FUNCTION_BLOCK FB_TCPModbusRequest
VAR_INPUT
	b_Enable: BOOL;
	str_IPAdress: STRING(15);
	
		
END_VAR
VAR_OUTPUT
	lreal_RealPower_kW:LREAL;
	lreal_Voltage_L1L2_V: LREAL;
	lreal_Voltage_L2L3_V: LREAL;
	lreal_Voltage_L3L1_V: LREAL;
	lreal_Voltage_L1_V: LREAL;
	lreal_Voltage_L2_V: LREAL;
	lreal_Voltage_L3_V: LREAL;
	lreal_Current_L1_A: LREAL;
	lreal_Current_L2_A: LREAL;
	lreal_Current_L3_A: LREAL;
	lreal_PeakPowerDay_kW: LREAL;
	lreal_Power2_kW: LREAL;
	lreal_ReactivePower_kVAr: LREAL;
	lreal_PowerFactor: LREAL;
	lreal_Frequency_Hz: LREAL;
	lreal_Efficiency: LREAL;
	lreal_InternalTemperature_C: LREAL;
	lreal_IsolationResistance_MOhm: LREAL;
	b_MeterOnline: BOOL;
	lreal_GridVoltage_L1L2_V: LREAL;
	lreal_GridVoltage_L2L3_V: LREAL;
	lreal_GridVoltage_L3L1_V: LREAL;
	lreal_GridVoltage_L1_V: LREAL;
	lreal_GridVoltage_L2_V: LREAL;
	lreal_GridVoltage_L3_V: LREAL;
	lreal_GridCurrent_L1_A: LREAL;
	lreal_GridCurrent_L2_A: LREAL;
	lreal_GridCurrent_L3_A: LREAL;
	lreal_GridPower_kW: LREAL;
	lreal_GridReactivePower_kVAr: LREAL;
	lreal_GridPowerFactor: LREAL;
	lreal_GridFrequency_Hz: LREAL;
	lreal_GridEnergyDelivered_kWh: LREAL;
	lreal_GridEnergySupllied_kWh: LREAL;
	
END_VAR
VAR
	i_State:INT;
	FB_SocketConnect : FB_SocketConnect;
	hSocket : T_HSOCKET;
	FB_SocketSend : FB_SocketSend;
	FB_SocketReceive : FB_SocketReceive;
	byteSendString : ARRAY[1..12] OF BYTE;
	byteSendString_2 : ARRAY[1..12] OF BYTE;
	FB_CloseSockets: FB_SocketCloseAll;
	
	ton_TimeOut: Ton;
	ton_WaitforReconnect: Ton;
	ton_ConnectionEstablised: Ton;
	time_ReconnectTime:TIME:=T#30M;
	b_configured: BOOL;
	byteReceiveString : ARRAY[1..200] OF BYTE;
	FB_BYTE_TO_WORD_1 : FB_CV_BYTE_TO_WORD;
	FB_BYTE_TO_WORD_2 : FB_CV_BYTE_TO_WORD;
	FB_BYTE_TO_WORD_Test1 : FB_CV_BYTE_TO_WORD;
	FB_BYTE_TO_WORD_Test2 : FB_CV_BYTE_TO_WORD;
	FB_WORD_TO_INT : FB_CV_WORD_TO_INT;
	ton_WaitforNetxtRequest: Ton;
	ton_Wait: Ton;
	int_SuccessCounter: INT;
	int_ReconnectCounter: INT;
	int_ErrorCount: INT;
	fbConvertWordToDword		: FB_CV_WORD_TO_DWORD;			//Convert Word to Dword
	fbConvertWordToDint			:	FB_CV_WORD_TO_DINT;
	fb_ConvertBytesToLreal		:fb_Convert4BytesToLreal;
	word1: WORD;
	x: INT;
END_VAR





IF NOT b_Enable THEN			// go to state 0 if not enabled
	i_State := 0;
END_IF


CASE i_State OF
	0:	// wait for enable state
		IF b_Enable THEN
			i_State := 1;
		END_IF
		FB_SocketConnect.bExecute := FALSE;
		FB_SocketSend.bExecute := FALSE;
		FB_SocketSend.bExecute := FALSE;
		ton_TimeOut.IN :=FALSE;	
		ton_ConnectionEstablised.IN := FALSE;
	

	1: // check if configured
		IF b_configured = FALSE THEN
			// request FC3, Register 32064, 25 Words 
			byteSendString[1] := 0;
			byteSendString[2] := 1;
			byteSendString[3] := 0;
			byteSendString[4] := 0;
			byteSendString[5] := 0;
			byteSendString[6] := 6;
			byteSendString[7] := 1;
			byteSendString[8] := 3;
			byteSendString[9] := 125;
			byteSendString[10] := 64;
			byteSendString[11] := 0;
			byteSendString[12] := 25;

			// request FC3, Register 37100 16#90EC, 25 Words 
			byteSendString_2[1] := 0;
			byteSendString_2[2] := 1;
			byteSendString_2[3] := 0;
			byteSendString_2[4] := 0;
			byteSendString_2[5] := 0;
			byteSendString_2[6] := 6;
			byteSendString_2[7] := 1;
			byteSendString_2[8] := 3;
			byteSendString_2[9] := 16#90;
			byteSendString_2[10] := 16#EC;
			byteSendString_2[11] := 0;
			byteSendString_2[12] := 38;
		
			b_configured := TRUE;
		END_IF
		i_State := i_State+1;
		
	2: // open socket
		FB_SocketConnect.bExecute := TRUE;
		ton_TimeOut.IN :=TRUE;
		i_State := i_State+1;
		
	3: // wait for connection established	
		IF NOT FB_SocketConnect.bBusy AND NOT FB_SocketConnect.bError THEN
			ton_TimeOut.IN :=FALSE;
			ton_ConnectionEstablised.IN := TRUE;
			i_State := i_State+1;
		ELSIF FB_SocketConnect.bError OR ton_TimeOut.Q THEN
			ton_TimeOut.IN :=FALSE;
			i_State := 100;
		END_IF
	
	4: //connection established, request data
		ton_Wait.IN := TRUE;
		FB_SocketSend.pSrc:= ADR( byteSendString ); 
			IF ton_Wait.Q THEN
			FB_SocketSend.bExecute := TRUE;
			ton_TimeOut.IN :=TRUE;
			ton_Wait.IN := FALSE;
			i_State := i_State+1;
		END_IF
	
	5: // wait for request sent
		IF NOT FB_SocketSend.bBusy AND NOT FB_SocketSend.bError THEN
			ton_TimeOut.IN :=FALSE;
			FB_SocketSend.bExecute := FALSE;
			i_State := i_State+1;  
		ELSIF FB_SocketSend.bError OR ton_TimeOut.Q THEN
			FB_SocketSend.bExecute := FALSE;
			ton_TimeOut.IN :=FALSE;
			i_State := 100;
		END_IF
		
	6: // wait for data
		ton_Wait.IN := TRUE;
		IF ton_Wait.Q THEN
			FB_SocketReceive.bExecute := TRUE;
			ton_Wait.IN := FALSE;
			i_State := i_State+1; 
		END_IF		 
	
	7:	
		ton_Wait.IN := TRUE;
		IF ton_Wait.Q THEN
			ton_TimeOut.IN :=TRUE;
			i_State := i_State+1; 
		END_IF	
	
	8: // convert received data
		IF NOT FB_SocketReceive.bBusy AND NOT FB_SocketReceive.bError THEN
			int_SuccessCounter := int_SuccessCounter+1;
			ton_TimeOut.IN :=FALSE;
			FB_SocketReceive.bExecute := FALSE;
	
			FB_BYTE_TO_WORD_1(byInputValue_1 := byteReceiveString[14],byInputValue_2 := byteReceiveString[15], Ebyteorderforconvert := Ebyteorder.EBIGENDIAN, woutputvalue => );
			lreal_Voltage_L1L2_V := WORD_TO_LREAL(FB_BYTE_TO_WORD_1.woutputvalue)/10;
			FB_BYTE_TO_WORD_1(byInputValue_1 := byteReceiveString[16],byInputValue_2 := byteReceiveString[17], Ebyteorderforconvert := Ebyteorder.EBIGENDIAN, woutputvalue => );
			lreal_Voltage_L2L3_V := WORD_TO_LREAL(FB_BYTE_TO_WORD_1.woutputvalue)/10;
			FB_BYTE_TO_WORD_1(byInputValue_1 := byteReceiveString[18],byInputValue_2 := byteReceiveString[19], Ebyteorderforconvert := Ebyteorder.EBIGENDIAN, woutputvalue => );
			lreal_Voltage_L3L1_V := WORD_TO_LREAL(FB_BYTE_TO_WORD_1.woutputvalue)/10;
			FB_BYTE_TO_WORD_1(byInputValue_1 := byteReceiveString[20],byInputValue_2 := byteReceiveString[21], Ebyteorderforconvert := Ebyteorder.EBIGENDIAN, woutputvalue => );
			lreal_Voltage_L1_V := WORD_TO_LREAL(FB_BYTE_TO_WORD_1.woutputvalue)/10;
			FB_BYTE_TO_WORD_1(byInputValue_1 := byteReceiveString[22],byInputValue_2 := byteReceiveString[23], Ebyteorderforconvert := Ebyteorder.EBIGENDIAN, woutputvalue => );
			lreal_Voltage_L2_V := WORD_TO_LREAL(FB_BYTE_TO_WORD_1.woutputvalue)/10;
			FB_BYTE_TO_WORD_1(byInputValue_1 := byteReceiveString[24],byInputValue_2 := byteReceiveString[25], Ebyteorderforconvert := Ebyteorder.EBIGENDIAN, woutputvalue => );
			lreal_Voltage_L3_V := WORD_TO_LREAL(FB_BYTE_TO_WORD_1.woutputvalue)/10;


			fb_ConvertBytesToLreal(	by_InputValue_1:= byteReceiveString[10], 
									by_InputValue_2:= byteReceiveString[11], 
									by_InputValue_3:= byteReceiveString[12], 
									by_InputValue_4:= byteReceiveString[13], 
									int_Divider:= 1000, 
									lreal_Output=> lreal_RealPower_kW);

			fb_ConvertBytesToLreal(	by_InputValue_1:= byteReceiveString[26], 
									by_InputValue_2:= byteReceiveString[27], 
									by_InputValue_3:= byteReceiveString[28], 
									by_InputValue_4:= byteReceiveString[29], 
									int_Divider:= 1000, 
									lreal_Output=> lreal_Current_L1_A);
									
			fb_ConvertBytesToLreal(	by_InputValue_1:= byteReceiveString[30], 
									by_InputValue_2:= byteReceiveString[31], 
									by_InputValue_3:= byteReceiveString[32], 
									by_InputValue_4:= byteReceiveString[33], 
									int_Divider:= 1000, 
									lreal_Output=> lreal_Current_L2_A);

			fb_ConvertBytesToLreal(	by_InputValue_1:= byteReceiveString[34], 
									by_InputValue_2:= byteReceiveString[35], 
									by_InputValue_3:= byteReceiveString[36], 
									by_InputValue_4:= byteReceiveString[37], 
									int_Divider:= 1000, 
									lreal_Output=> lreal_Current_L3_A);
									
			fb_ConvertBytesToLreal(	by_InputValue_1:= byteReceiveString[38], 
									by_InputValue_2:= byteReceiveString[39], 
									by_InputValue_3:= byteReceiveString[40], 
									by_InputValue_4:= byteReceiveString[41], 
									int_Divider:= 1000, 
									lreal_Output=> lreal_PeakPowerDay_kW );

			fb_ConvertBytesToLreal(	by_InputValue_1:= byteReceiveString[42], 
									by_InputValue_2:= byteReceiveString[43], 
									by_InputValue_3:= byteReceiveString[44], 
									by_InputValue_4:= byteReceiveString[45], 
									int_Divider:= 1000, 
									lreal_Output=> lreal_Power2_kW);
			
			fb_ConvertBytesToLreal(	by_InputValue_1:= byteReceiveString[46], 
									by_InputValue_2:= byteReceiveString[47], 
									by_InputValue_3:= byteReceiveString[48], 
									by_InputValue_4:= byteReceiveString[49], 
									int_Divider:= 1000, 
									lreal_Output=>lreal_ReactivePower_kVAr );

			FB_BYTE_TO_WORD_1(byInputValue_1 := byteReceiveString[50],byInputValue_2 := byteReceiveString[51], Ebyteorderforconvert := Ebyteorder.EBIGENDIAN, woutputvalue => );
			lreal_PowerFactor := WORD_TO_LREAL(FB_BYTE_TO_WORD_1.woutputvalue)/1000;
			FB_BYTE_TO_WORD_1(byInputValue_1 := byteReceiveString[52],byInputValue_2 := byteReceiveString[53], Ebyteorderforconvert := Ebyteorder.EBIGENDIAN, woutputvalue => );
			lreal_Frequency_Hz := WORD_TO_LREAL(FB_BYTE_TO_WORD_1.woutputvalue)/100;
			FB_BYTE_TO_WORD_1(byInputValue_1 := byteReceiveString[54],byInputValue_2 := byteReceiveString[55], Ebyteorderforconvert := Ebyteorder.EBIGENDIAN, woutputvalue => );
			lreal_Efficiency := WORD_TO_LREAL(FB_BYTE_TO_WORD_1.woutputvalue)/100;
			FB_BYTE_TO_WORD_1(byInputValue_1 := byteReceiveString[56],byInputValue_2 := byteReceiveString[57], Ebyteorderforconvert := Ebyteorder.EBIGENDIAN, woutputvalue => );
			lreal_InternalTemperature_C := WORD_TO_LREAL(FB_BYTE_TO_WORD_1.woutputvalue)/10;
			FB_BYTE_TO_WORD_1(byInputValue_1 := byteReceiveString[58],byInputValue_2 := byteReceiveString[59], Ebyteorderforconvert := Ebyteorder.EBIGENDIAN, woutputvalue => );
			lreal_IsolationResistance_MOhm := WORD_TO_LREAL(FB_BYTE_TO_WORD_1.woutputvalue)/1000;

		
			//FB_WORD_TO_INT(wInputValue := FB_BYTE_TO_WORD.woutputvalue, iOutputValue => );
			//lreal_RealPower_kW := (INT_TO_LREAL(FB_WORD_TO_INT.iOutputValue))/1000;
			i_State := 15; //i_State+1;
		ELSIF FB_SocketSend.bError OR ton_TimeOut.Q THEN
 			FB_SocketReceive.bExecute := FALSE;
			ton_TimeOut.IN :=FALSE;
			i_State := 100;
		END_IF

	15: // close sockets
		FB_CloseSockets.bExecute := TRUE;
		ton_TimeOut.IN :=TRUE;
		i_State := i_State+1;
		
	16: // wait for sockets closed
		
		IF NOT FB_CloseSockets.bBusy THEN
			int_ReconnectCounter := int_ReconnectCounter+1;
			FB_CloseSockets.bExecute := FALSE;
			i_State := 0;
		ELSIF FB_CloseSockets.bError THEN
			int_ReconnectCounter := int_ReconnectCounter+1;
			FB_CloseSockets.bExecute := FALSE;
			i_State := 0;
		END_IF
	
	17: // open socket
		FB_SocketConnect.bExecute := TRUE;
		ton_TimeOut.IN :=TRUE;
		i_State := i_State+1;
		
	18: // wait for connection established	
		IF NOT FB_SocketConnect.bBusy AND NOT FB_SocketConnect.bError THEN
			ton_TimeOut.IN :=FALSE;
			ton_ConnectionEstablised.IN := TRUE;
			i_State := 20;
		ELSIF FB_SocketConnect.bError OR ton_TimeOut.Q THEN
			ton_TimeOut.IN :=FALSE;
			i_State := 100;
		END_IF
	
	20: //connection established, request data second poll
		ton_Wait.IN := TRUE;
		FB_SocketSend.pSrc:= ADR( byteSendString_2 ); 
			IF ton_Wait.Q THEN
			FB_SocketSend.bExecute := TRUE;
			ton_TimeOut.IN :=TRUE;
			ton_Wait.IN := FALSE;
			i_State := i_State+1;
		END_IF
	
	21: // wait for request sent
		IF NOT FB_SocketSend.bBusy AND NOT FB_SocketSend.bError THEN
			ton_TimeOut.IN :=FALSE;
			FB_SocketSend.bExecute := FALSE;
			x:=x+1;
			i_State := i_State+1;  
		ELSIF FB_SocketSend.bError OR ton_TimeOut.Q THEN
			FB_SocketSend.bExecute := FALSE;
			ton_TimeOut.IN :=FALSE;
			x:=x-10;
			i_State := 100;
		END_IF
		
	22: // wait for data
		ton_Wait.IN := TRUE;
		IF ton_Wait.Q THEN
			FB_SocketReceive.bExecute := TRUE;
			ton_Wait.IN := FALSE;
			i_State := i_State+1; 
		END_IF		 
	
	23:	
		ton_Wait.IN := TRUE;
		IF ton_Wait.Q THEN
			ton_TimeOut.IN :=TRUE;
			i_State := i_State+1; 
		END_IF	
	
	24: // convert received data
		IF NOT FB_SocketReceive.bBusy AND NOT FB_SocketReceive.bError THEN
			int_SuccessCounter := int_SuccessCounter+1;
			ton_TimeOut.IN :=FALSE;
			FB_SocketReceive.bExecute := FALSE;
	
			FB_BYTE_TO_WORD_1(byInputValue_1 := byteReceiveString[10],byInputValue_2 := byteReceiveString[11], Ebyteorderforconvert := Ebyteorder.EBIGENDIAN, woutputvalue => );
			IF WORD_TO_LREAL(FB_BYTE_TO_WORD_1.woutputvalue) = 0 THEN
				b_MeterOnline :=FALSE;
			ELSIF WORD_TO_LREAL(FB_BYTE_TO_WORD_1.woutputvalue) = 1 THEN
				b_MeterOnline :=TRUE;
			END_IF
			
			fb_ConvertBytesToLreal(	by_InputValue_1:= byteReceiveString[12], 
									by_InputValue_2:= byteReceiveString[13], 
									by_InputValue_3:= byteReceiveString[14], 
									by_InputValue_4:= byteReceiveString[15], 
									int_Divider:= 10, 
									lreal_Output=> lreal_GridVoltage_L1_V );
									
			fb_ConvertBytesToLreal(	by_InputValue_1:= byteReceiveString[16], 
									by_InputValue_2:= byteReceiveString[17], 
									by_InputValue_3:= byteReceiveString[18], 
									by_InputValue_4:= byteReceiveString[19], 
									int_Divider:= 10, 
									lreal_Output=> lreal_GridVoltage_L2_V);
									
			fb_ConvertBytesToLreal(	by_InputValue_1:= byteReceiveString[20], 
									by_InputValue_2:= byteReceiveString[21], 
									by_InputValue_3:= byteReceiveString[22], 
									by_InputValue_4:= byteReceiveString[23], 
									int_Divider:= 10, 
									lreal_Output=> lreal_GridVoltage_L3_V);
								
			fb_ConvertBytesToLreal(	by_InputValue_1:= byteReceiveString[24], 
									by_InputValue_2:= byteReceiveString[25], 
									by_InputValue_3:= byteReceiveString[26], 
									by_InputValue_4:= byteReceiveString[27], 
									int_Divider:= 100, 
									lreal_Output=> lreal_GridCurrent_L1_A );
									
			fb_ConvertBytesToLreal(	by_InputValue_1:= byteReceiveString[24], 
									by_InputValue_2:= byteReceiveString[25], 
									by_InputValue_3:= byteReceiveString[26], 
									by_InputValue_4:= byteReceiveString[27], 
									int_Divider:= 100, 
									lreal_Output=> lreal_GridCurrent_L1_A );
									
			fb_ConvertBytesToLreal(	by_InputValue_1:= byteReceiveString[28], 
									by_InputValue_2:= byteReceiveString[29], 
									by_InputValue_3:= byteReceiveString[30], 
									by_InputValue_4:= byteReceiveString[31], 
									int_Divider:= 100, 
									lreal_Output=> lreal_GridCurrent_L2_A );
									
			fb_ConvertBytesToLreal(	by_InputValue_1:= byteReceiveString[32], 
									by_InputValue_2:= byteReceiveString[33], 
									by_InputValue_3:= byteReceiveString[34], 
									by_InputValue_4:= byteReceiveString[35], 
									int_Divider:= 100, 
									lreal_Output=> lreal_GridCurrent_L3_A );
									
			fb_ConvertBytesToLreal(	by_InputValue_1:= byteReceiveString[36], 
									by_InputValue_2:= byteReceiveString[37], 
									by_InputValue_3:= byteReceiveString[38], 
									by_InputValue_4:= byteReceiveString[39], 
									int_Divider:= 1000, 
									lreal_Output=> lreal_GridPower_kW);
									
			fb_ConvertBytesToLreal(	by_InputValue_1:= byteReceiveString[40], 
									by_InputValue_2:= byteReceiveString[41], 
									by_InputValue_3:= byteReceiveString[42], 
									by_InputValue_4:= byteReceiveString[43], 
									int_Divider:= 1000, 
									lreal_Output=> lreal_GridReactivePower_kVAr);
											
			//FB_BYTE_TO_WORD_1(byInputValue_1 := byteReceiveString[44],byInputValue_2 := byteReceiveString[45], Ebyteorderforconvert := Ebyteorder.EbigENDIAN, woutputvalue => );
			//lreal_GridPowerFactor := WORD_TO_LREAL(FB_BYTE_TO_WORD_1.woutputvalue)/1000;

			lreal_GridPowerFactor := INT_TO_LREAL(WORD_TO_INT((SHL(BYTE_TO_WORD(byteReceiveString[44]),8) + BYTE_TO_WORD(byteReceiveString[45]))))/1000;


		
			FB_BYTE_TO_WORD_1(byInputValue_1 := byteReceiveString[46],byInputValue_2 := byteReceiveString[47], Ebyteorderforconvert := Ebyteorder.EbigENDIAN, woutputvalue => );
			lreal_GridFrequency_Hz := WORD_TO_LREAL(FB_BYTE_TO_WORD_1.woutputvalue)/100;
			
			fb_ConvertBytesToLreal(	by_InputValue_1:= byteReceiveString[48], 
									by_InputValue_2:= byteReceiveString[49], 
									by_InputValue_3:= byteReceiveString[50], 
									by_InputValue_4:= byteReceiveString[51], 
									int_Divider:= 100, 
									lreal_Output=> lreal_GridEnergyDelivered_kWh);
									
			fb_ConvertBytesToLreal(	by_InputValue_1:= byteReceiveString[52], 
									by_InputValue_2:= byteReceiveString[53], 
									by_InputValue_3:= byteReceiveString[54], 
									by_InputValue_4:= byteReceiveString[55], 
									int_Divider:= 100, 
									lreal_Output=> lreal_GridEnergySupllied_kWh );
			
			fb_ConvertBytesToLreal(	by_InputValue_1:= byteReceiveString[62], 
									by_InputValue_2:= byteReceiveString[63], 
									by_InputValue_3:= byteReceiveString[64], 
									by_InputValue_4:= byteReceiveString[65], 
									int_Divider:= 10 , 
									lreal_Output=> lreal_GridVoltage_L1L2_V);

			fb_ConvertBytesToLreal(	by_InputValue_1:= byteReceiveString[66], 
									by_InputValue_2:= byteReceiveString[67], 
									by_InputValue_3:= byteReceiveString[68], 
									by_InputValue_4:= byteReceiveString[69], 
									int_Divider:= 10 , 
									lreal_Output=> lreal_GridVoltage_L2L3_V);

			fb_ConvertBytesToLreal(	by_InputValue_1:= byteReceiveString[70], 
									by_InputValue_2:= byteReceiveString[71], 
									by_InputValue_3:= byteReceiveString[72], 
									by_InputValue_4:= byteReceiveString[73], 
									int_Divider:= 10 , 
									lreal_Output=> lreal_GridVoltage_L3L1_V);

	
			i_State := 30; //i_State+1;
		ELSIF FB_SocketSend.bError OR ton_TimeOut.Q THEN
			FB_SocketReceive.bExecute := FALSE;
			ton_TimeOut.IN :=FALSE;
			i_State := 100;
		END_IF

	
	30: // for for next request
		ton_Wait.IN :=FALSE;
		ton_WaitforNetxtRequest.IN := TRUE;
		IF NOT b_Enable THEN
			ton_WaitforNetxtRequest.IN := FALSE;
			i_State := 40;
		END_IF
		IF ton_WaitforNetxtRequest.Q THEN
			ton_WaitforNetxtRequest.IN := FALSE;
			i_State := 4;
		END_IF
		IF 	ton_ConnectionEstablised.Q THEN 
			ton_WaitforNetxtRequest.IN := FALSE;
			i_State := 40;
		END_IF

	40: // close sockets
		FB_CloseSockets.bExecute := TRUE;
		ton_TimeOut.IN :=TRUE;
		i_State := i_State+1;
		
	41: // wait for sockets closed
		
		IF NOT FB_CloseSockets.bBusy THEN
			int_ReconnectCounter := int_ReconnectCounter+1;
			FB_CloseSockets.bExecute := FALSE;
			i_State := 0;
		ELSIF FB_CloseSockets.bError THEN
			int_ReconnectCounter := int_ReconnectCounter+1;
			FB_CloseSockets.bExecute := FALSE;
			i_State := 0;
		END_IF



	100: // wait state for reconect
		
		FB_SocketConnect.bExecute := FALSE;
		FB_SocketSend.bExecute := FALSE;
		FB_SocketReceive.bExecute := FALSE;
		ton_ConnectionEstablised.IN := FALSE;
		ton_Wait.IN :=FALSE;
		ton_TimeOut.IN :=FALSE;
		ton_WaitforReconnect.IN := TRUE;
		IF ton_WaitforReconnect.Q THEN
			int_ErrorCount := int_ErrorCount+1;
			ton_WaitforReconnect.IN := FALSE;
			i_State := 40;
		END_IF
	
END_CASE



FB_SocketConnect(
	sSrvNetId := '',
	sRemoteHost := str_IPAdress,
	nRemotePort := 502,
	bExecute := ,
	tTimeout := T#1S,
	bBusy =>,
	bError =>,
	nErrId =>,
	hSocket => hSocket);
	
FB_SocketSend(
	sSrvNetId:= '', 
	hSocket:= hSocket, 
	cbLen:= 12,
	pSrc:= , //ADR( byteSendString ), 
	bExecute:= , 
	tTimeout:= T#3S, 
	bBusy=> , 
	bError=> , 
	nErrId=> );
	
FB_SocketReceive(
	sSrvNetId:= '', 
	hSocket:= hSocket, 
	cbLen:= 200, 
	pDest:= ADR( byteReceiveString ), 
	bExecute:= , 
	tTimeout:= T#3S, 
	bBusy=> , 
	bError=> , 
	nErrId=> , 
	nRecBytes=> );

FB_CloseSockets(
	sSrvNetId:= '', 
	bExecute:= , 
	tTimeout:= T#2S, 
	bBusy=> , 
	bError=> , 
	nErrId=> );
	
ton_TimeOut(PT := T#5S);
ton_WaitforReconnect(PT := T#10S);
ton_ConnectionEstablised(pt := time_ReconnectTime);
ton_WaitforNetxtRequest(PT:= T#10S);
ton_Wait(PT:=T#2S);

END_FUNCTION_BLOCK

(* stored: Version 1.1.0.1, ProductVersion 3.1.4024.11
   POU FB_TCPModbusRequest: Id {e4dd9c52-662d-43eb-bfd3-6aec585bcd8d}, SpecialFunc None *)
